# EPICS substitutions: old/bl6-SkfChopper/bl6-SkfChopperApp/Db/hexaDskScanAssist_saveRst.substitutions
file save_restoreStatus.db
{
pattern {P}
       {BL6:SavRst:ChopSkfCalc16:}
}
